// TIA Portal V17 export
// export: Created 2025-03-07T09:18:28.178798Z, ExportSetting WithDefaults, DisplayName Totally Integrated Automation Portal, DisplayVersion V17 Update 8, DisplayName TIA Portal Openness, DisplayVersion V17 Update 8, DisplayName TIA Portal Version Control Interface, DisplayVersion V17, DisplayName SINAMICS Startdrive Advanced, DisplayVersion V17 SP2, DisplayName SINAMICS Startdrive G110M, G120, G120C, G120D, G120P, G115D, DisplayVersion V17 SP2, DisplayName SINAMICS Startdrive G130, G150, S120, S150, SINAMICS MV, S210, DisplayVersion V17 SP2, DisplayName STEP 7 Professional, DisplayVersion V17 Update 8, DisplayName SINUMERIK ONE STEP 7 Toolbox, DisplayVersion V17 Update 12, DisplayName SINUMERIK 840D sl STEP 7 Toolbox, DisplayVersion V17 Update 12, DisplayName STEP 7 Safety, DisplayVersion V17 Update 6, DisplayName WinCC Advanced, DisplayVersion V17 Update 8
FUNCTION "FC505_SETUP_DECODING" : Void   // FC505, LAD
{ S7_Optimized_Access := 'FALSE' }
AUTHOR : ETXETAR
VERSION : 1.0
// stored: AutoNumber false, IsIECCheckEnabled false, SetENOAutomatically false, UDAEnableTagReadback false
   VAR_TEMP
      RETVAL : Int;
   END_VAR
   VAR_TEMP   // added for the SCL form of the ladder/FBD networks
      _w1 : Bool;
      _w2 : Bool;
   END_VAR
BEGIN

REGION Network 1: SETUP 1
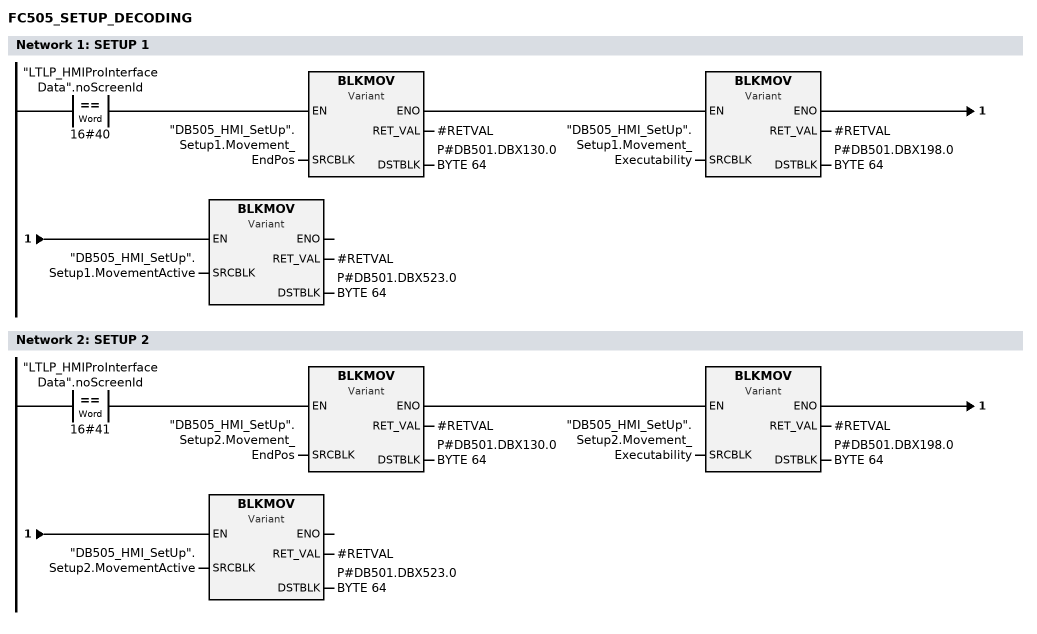
   RUNG wire#powerrail
      { S7_Templates := "SrcType := Word" } EQ_Contact(in1 := "LTLP_HMIProInterfaceData".noScreenId, in2 := 16#40)
      { S7_Templates := "blk_type := Variant" } BLKMOV(SRCBLK := "DB505_HMI_SetUp".Setup1.Movement_EndPos, RET_VAL => #RETVAL, DSTBLK => P#DB501.DBX130.0 BYTE 64)
      { S7_Templates := "blk_type := Variant" } BLKMOV(SRCBLK := "DB505_HMI_SetUp".Setup1.Movement_Executability, RET_VAL => #RETVAL, DSTBLK => P#DB501.DBX198.0 BYTE 64)
      { S7_Templates := "blk_type := Variant" } BLKMOV(SRCBLK := "DB505_HMI_SetUp".Setup1.MovementActive, RET_VAL => #RETVAL, DSTBLK => P#DB501.DBX523.0 BYTE 64)
   END_RUNG
   // the same network as SCL:
   #RETVAL := BLKMOV(EN := "LTLP_HMIProInterfaceData".noScreenId = 16#40,
                     SRCBLK := "DB505_HMI_SetUp".Setup1.Movement_EndPos,
                     DSTBLK => P#DB501.DBX130.0 BYTE 64,
                     ENO => #_w1);
   #RETVAL := BLKMOV(EN := #_w1,
                     SRCBLK := "DB505_HMI_SetUp".Setup1.Movement_Executability,
                     DSTBLK => P#DB501.DBX198.0 BYTE 64,
                     ENO => #_w2);
   IF #_w2 THEN
       #RETVAL := BLKMOV(SRCBLK := "DB505_HMI_SetUp".Setup1.MovementActive, DSTBLK => P#DB501.DBX523.0 BYTE 64);
   END_IF;
END_REGION

REGION Network 2: SETUP 2
   RUNG wire#powerrail
      { S7_Templates := "SrcType := Word" } EQ_Contact(in1 := "LTLP_HMIProInterfaceData".noScreenId, in2 := 16#41)
      { S7_Templates := "blk_type := Variant" } BLKMOV(SRCBLK := "DB505_HMI_SetUp".Setup2.Movement_EndPos, RET_VAL => #RETVAL, DSTBLK => P#DB501.DBX130.0 BYTE 64)
      { S7_Templates := "blk_type := Variant" } BLKMOV(SRCBLK := "DB505_HMI_SetUp".Setup2.Movement_Executability, RET_VAL => #RETVAL, DSTBLK => P#DB501.DBX198.0 BYTE 64)
      { S7_Templates := "blk_type := Variant" } BLKMOV(SRCBLK := "DB505_HMI_SetUp".Setup2.MovementActive, RET_VAL => #RETVAL, DSTBLK => P#DB501.DBX523.0 BYTE 64)
   END_RUNG
   // the same network as SCL:
   #RETVAL := BLKMOV(EN := "LTLP_HMIProInterfaceData".noScreenId = 16#41,
                     SRCBLK := "DB505_HMI_SetUp".Setup2.Movement_EndPos,
                     DSTBLK => P#DB501.DBX130.0 BYTE 64,
                     ENO => #_w1);
   #RETVAL := BLKMOV(EN := #_w1,
                     SRCBLK := "DB505_HMI_SetUp".Setup2.Movement_Executability,
                     DSTBLK => P#DB501.DBX198.0 BYTE 64,
                     ENO => #_w2);
   IF #_w2 THEN
       #RETVAL := BLKMOV(SRCBLK := "DB505_HMI_SetUp".Setup2.MovementActive, DSTBLK => P#DB501.DBX523.0 BYTE 64);
   END_IF;
END_REGION
END_FUNCTION
